(* CODESYS project CmpEmiconLCD.library
   Title: LCD Services
   Author: Emicon
   DefaultNamespace: EmLCD
   Version: 3.5.13.0
   Company: Emicon

Project tree, tasks and I/O mapping:
  function lcd_puts [ST]
  function get_current_screen [ST]
  function display_screen [ST]
  function set_default_screen [ST]
  function get_default_screen [ST]
  function set_visibility [ST]
  global variables GVL
  function menu_item_create [ST]
*)

// GVL
VAR_GLOBAL CONSTANT
	VISIBLE: BOOL := 0;
	HIDDEN: BOOL := 1; 
END_VAR

// lcd_puts
FUNCTION lcd_puts: INT
VAR_INPUT
	usiScreen : USINT;		// номер экрана 0-9
	iLine: USINT;			// Строка 0-1
	iPos: USINT;			// Столбец 0-249
	stData: STRING(251);	// Текст 1-250 сиволов
END_VAR
VAR	
END_VAR

END_FUNCTION

// get_current_screen
(*
 * Возвращает номер отображаемого экрана на LCD.
 *)
FUNCTION get_current_screen : usint
VAR_INPUT
END_VAR
VAR
END_VAR

END_FUNCTION

// display_screen
(*
 * Выводит на LCD экран с заданным номером.
 *)
FUNCTION display_screen : INT
VAR_INPUT
	n : USINT; // номер экрана
END_VAR
VAR
END_VAR

END_FUNCTION

// set_default_screen
(*
 * Устанавливает эран по умолчанию.
 *)
FUNCTION set_default_screen : USINT
VAR_INPUT
	n : USINT; // номер экрана
END_VAR
VAR
END_VAR

END_FUNCTION

// get_default_screen
(*
 * Возвращает номер экрана по умолчанию.
 *)
FUNCTION get_default_screen : usint
VAR_INPUT
END_VAR
VAR
END_VAR

END_FUNCTION

// set_visibility
(*
 * Установка видимости экрана.
 *)
FUNCTION set_visibility : int
VAR_INPUT
	n: USINT; // номер экрана
	visibility: BOOL;
END_VAR
VAR
END_VAR

END_FUNCTION

// menu_item_create
FUNCTION menu_item_create : UDINT
VAR_INPUT
	screen: USINT;			// номер экрана меню 0-9
	st_line1: STRING(251);	// Текст 1-250 сиволов
	st_line2: STRING(251);	// Текст 1-250 сиволов
	p_menu_function : POINTER TO BYTE; // указатель на функцию
	
END_VAR
VAR
END_VAR

END_FUNCTION
